PROGRAM P20_ExhaustFan
VAR
	(*****************Wentylator wyciągaowy*******************)
	QbExhaustSystemEnable					AT %Q*	:BOOL;		
	IbExhaustSystemSwitchNormalMode			AT %I*	:BOOL;		
	IbExhaustSystemSwitchExMode				AT %I*	:BOOL;		
	IbExhaustSystemReady					AT %I*	:BOOL;		
	IbExhaustSystemAlarm					AT %I*	:BOOL;		
	IbExhaustSystemFlowOk					AT %I*	:BOOL;		
	IbExhaustSystemAlarmLevel1				AT %I*	:BOOL;		
			
	fbSensorAirFlow							: FB_SensorFlow;
	
END_VAR


QbExhaustSystemEnable := VIS.bExEnableShow OR bExEnable;

aSensors();

ExSensorWarning[1].sDescription:='Alarm poziomu 1 detekcja gazu 10%DGW';
IF (IbExhaustSystemAlarmLevel1 AND QbExhaustSystemEnable) AND NOT ExSensorWarning[1].bWarning THEN
	ExSensorWarning[1].bWarning		:=	TRUE;
ELSIF ( NOT IbExhaustSystemAlarmLevel1 )AND ExSensorWarning[1].bAcknowledge THEN
	ExSensorWarning[1].bWarning		:=	FALSE;
	ExSensorWarning[1].bAcknowledge	:=	FALSE;
	VIS.uliWarningAcknowledge.24 	:=	FALSE;
ELSIF ExSensorWarning[1].bAcknowledge THEN
	ExSensorWarning[1].bAcknowledge	:=	TRUE;
END_IF


ExhaustFanError;
IF ExhaustFanError.bReset THEN
	ExhaustFanError.bError				:= FALSE;
	ExhaustFanError.udiStationID		:= 0;
	ExhaustFanError.nErrorCode			:= 0;
	ExhaustFanError.bReset				:= FALSE;
	ExhaustFanError.sErrorString		:= '';
	ExhaustFanError.sErrorString2		:= '';	
END_IF
IF IbExhaustSystemAlarm AND QbExhaustSystemEnable AND NOT VIS.bErrorOccure THEN
	ExhaustFanError.bError				:= TRUE;
	ExhaustFanError.udiStationID		:= 75;
	ExhaustFanError.nErrorCode			:= 372;
	ExhaustFanError.bReset				:= FALSE;
	ExhaustFanError.sErrorString		:= 'System wentylacji Ex - błąd - sprawdź szafę R4 Ex';
	ExhaustFanError.sErrorString2		:= '';
ELSIF NOT QbExhaustSystemEnable THEN
	ExhaustFanError.bError				:= FALSE;
END_IF

ACTION aSensors:
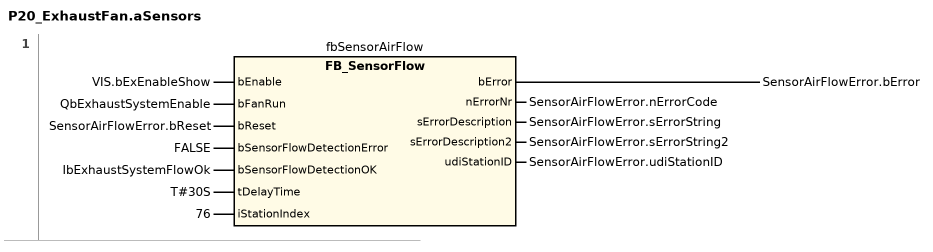
// NETWORK 1
fbSensorAirFlow(
    bEnable := VIS.bExEnableShow,
    bFanRun := QbExhaustSystemEnable,
    bReset := SensorAirFlowError.bReset,
    bSensorFlowDetectionError := FALSE,
    bSensorFlowDetectionOK := IbExhaustSystemFlowOk,
    tDelayTime := T#30S,
    iStationIndex := 76,
    nErrorNr => SensorAirFlowError.nErrorCode,
    sErrorDescription => SensorAirFlowError.sErrorString,
    sErrorDescription2 => SensorAirFlowError.sErrorString2,
    udiStationID => SensorAirFlowError.udiStationID); // FB_SensorFlow
SensorAirFlowError.bError := fbSensorAirFlow.bError;
END_ACTION

END_PROGRAM

(* stored: Version 1.1.0.1, ProductVersion 3.1.4026.13, FileIdentifier 74b77718c2c444994bc279109428e3d0ca51e3c8, FileSignature a6bf0707e109eeba772a0a5c0fb0b2ca927517d5723863eec261e65fc38ebf5210ece64ad16ad62593d32896d968fce0e35b90de2b5c3061cf8f8b865c9c5c7a9a31a8dea079201b48db55e563cc196e681ba41a0232fc5c96db7cd2d09f9d265161fe6f53e20ecb7f3e402449194aaaa22869ecead9b1e2fd7628dacdde1398ebbfd4cadddcb028f4cc624c24e878b63b19aff87253d5a42d363324036d4957dc04ae15f402e63b64ab8b8ab3532190a6ef6c6f6f6df1a7206a77a3f8292b1368f10ad1b724415bdab1b59d8da7f90dc1d8adabbb49009257c950038b9be7c93524fa6c4c10289bd085f94a9c51b24e9d5ec91261699886cbb585edbe226428
   POU P20_ExhaustFan: Id {812e0fd8-628b-45d6-b5b7-23d705c3fcbe}, SpecialFunc None
   Action aSensors: Id {f604fdf9-3200-4d58-8974-62b91f4ebfba} *)
